// TwinCAT 3 PLC project Plc
// ProgramVersion: 3.1.4024.0
// libraries:
//   CmpBitmapPool, * (System)
//   Tc2_Standard, * (Beckhoff Automation GmbH)
//   Tc2_System, * (Beckhoff Automation GmbH)
//   Tc3_Module, * (Beckhoff Automation GmbH)
//   VisuDialogs, * (System)
//   VisuSymbols,3.5.10.0,System
// project tree:
//   / Gestore di visualizzazione.TcVMO (not stored), GlobalTextList.TcGTLO, ImagePool.TcIPO (not stored), PlcTask.TcTTO
//   GVLs/ GVL.TcGVL
//   POUs/ MAIN.TcPOU
//   VISUs/ Visualization.TcVIS
// real-time tasks:
//   TASK PlcTask: cycle T#10ms, priority 20, ADS port 350

CONFIGURATION Plc
    RESOURCE PLC ON TwinCAT3
        TASK PlcTask(INTERVAL := T#10ms, PRIORITY := 20);
        PROGRAM MAIN WITH PlcTask : MAIN;
    END_RESOURCE
END_CONFIGURATION

// ---- GVLs/GVL.TcGVL
{attribute 'qualified_only'}
VAR_GLOBAL
	//input
	PB1: BOOL;
	PB2: BOOL;
	PBE: BOOL;
	PS1: BOOL;
	PS2: BOOL;
	PS3: BOOL;
	PS4: BOOL;
	FS1: BOOL;
	FS2: BOOL;
	SB1: BOOL;
	SB2: BOOL;
	SB3: BOOL;
	LC1: REAL; //Valore di tensione da 0V a 10V (0 Kg - 15 Kg)
	
	//output
	L1: BOOL;
	L2: BOOL;
	L3: BOOL;
	L4: BOOL;
	L5: BOOL;
	M1 : BOOL;
	M2 : BOOL;
	M3 : BOOL;
	M4 : BOOL;
	M5 : BOOL;
END_VAR

// ---- POUs/MAIN.TcPOU
PROGRAM MAIN
VAR
END_VAR

END_PROGRAM

// ---- GlobalTextList.TcGTLO
TEXTLIST GlobalTextList
  809 = '%d'
  216 = '%f'
  890 = '%r'
  68 = 'Emergenza'
  801 = 'FS1'
  524 = 'FS2'
  765 = 'LC1'
  869 = 'M1'
  802 = 'M2'
  115 = 'M3'
  287 = 'M4'
  498 = 'M5'
  273 = 'PEso '
  564 = 'Peso Prosciutto'
  388 = 'PS1'
  762 = 'Ps1'
  310 = 'PS2'
  806 = 'PS3'
  525 = 'PS4'
  656 = 'SB1'
  665 = 'SB2'
  112 = 'SB3'
  871 = 'Start'
  275 = 'Stop'
END_TEXTLIST

// ---- VISUs/Visualization.TcVIS
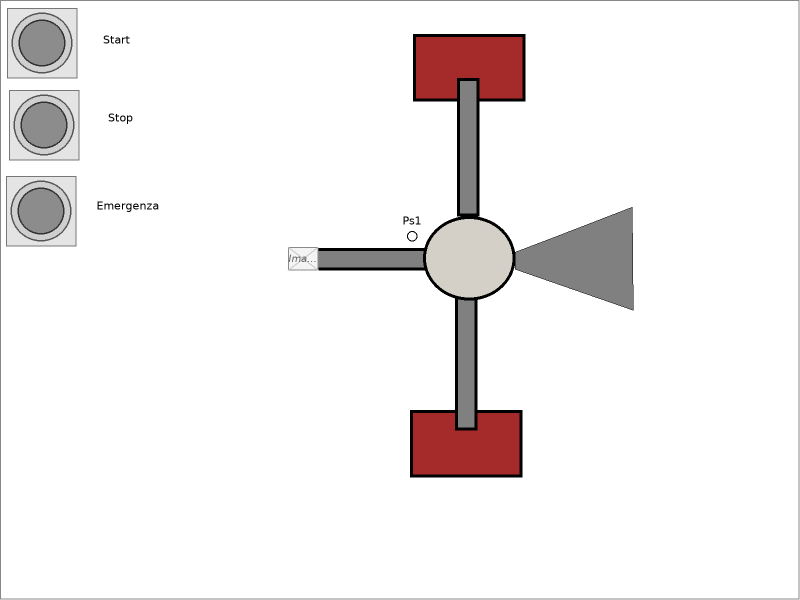
VISUALIZATION Visualization  // 800x600
    Rectangle (473,-103 67x112), angle 270
    Rectangle (470,273 67x112), angle 270
    Rectangle (856,994 145x265), angle 270
    PushSwitch (7,8 70x70), behaviour: TAP, style: Switch-PushSwitch-Gray
    Label (89,25 55x30), "Start"
    PushSwitch (9,90 70x70), behaviour: TAP, style: Switch-PushSwitch-Gray
    Label (88,103 65x30), "Stop"
    PushSwitch (6,176 70x70), behaviour: TAP, style: Switch-PushSwitch-Gray
    Label (83,191 90x30), "Emergenza"
    Rectangle (289,248 138x22)
    Rectangle (304,201 138x22), angle 90
    Rectangle (302,415 138x22), angle 90
    Ellipse (423,216 92x84)
    Polygon (515,252) (557,236) (632,207) (633,310) (515,269)
    Image (288,247 30x23), image: ImagePool.ham
    Ellipse (407,231 10x10), colour toggle: GVL.bPs1
    Label (388,215 48x12), "Ps1"
END_VISUALIZATION
